// TIA Portal V18 export
DATA_BLOCK "lightColumn_DB"   // DB48
VERSION : 0.1
// stored: AutoNumber true, DBAccessibleFromOPCUA true, InstanceOfName lightColumn, InstanceOfType FB
"lightColumn"
   // VAR_INPUT
   //    er : Bool;
   //    readyMan : Bool;
   //    runAuto : Bool;
   // END_VAR
   // VAR_OUTPUT
   //    green : Bool;
   //    red : Bool;
   //    orange : Bool;
   // END_VAR
BEGIN
END_DATA_BLOCK
